TYPE HMI_STS_RbtFanucUnloading EXTENDS HMI_STS_RbtFanuc:
STRUCT
	;//add custom on top of library block here
END_STRUCT
END_TYPE

(* stored: Version 1.1.0.1
   DUT HMI_STS_RbtFanucUnloading: Id {e3d0c409-98fc-42c3-bcd8-9169a66db4f2} *)
